// TIA Portal V15.1 export
// export: Created 2024-06-21T08:40:46.3013214Z, ExportSetting WithDefaults, DisplayName Totally Integrated Automation Portal, DisplayVersion V15.1 Update 5, DisplayName TIA Portal Openness, DisplayVersion V15.1 Update 5, DisplayName SINAMICS Startdrive Advanced, DisplayVersion V15.1, DisplayName G130, G150, S120, S150, SINAMICS MV, S210, DisplayVersion V15.1, DisplayName G110M, G120, G120C, G120D, G120P, DisplayVersion V15.1, DisplayName STEP 7 Professional, DisplayVersion V15.1 Update 5, DisplayName STEP 7 Safety, DisplayVersion V15.1, DisplayName WinCC Professional, DisplayVersion V15.1 Update 5, DisplayName SIMATIC Visualization Architect, DisplayVersion V15.1
DATA_BLOCK "_209210NCB02TagSeq"   // DB1620
{ S7_Optimized_Access := 'TRUE' }
VERSION : 0.1
// stored: AutoNumber false, DBAccessibleFromOPCUA true, InstanceOfName 209210NCB02TagSeq, InstanceOfType FB
"209210NCB02TagSeq"
   // // inherited from GRAPH_BASE
   // VAR
   //    OFF_SQ_BASE : Bool;
   // END_VAR
   // VAR_INPUT
   //    OFF_SQ { ExternalWritable := 'False'} : Bool;
   //    INIT_SQ { ExternalWritable := 'False'} : Bool;
   //    ACK_EF { ExternalWritable := 'False'} : Bool;
   //    S_PREV { ExternalWritable := 'False'} : Bool;
   //    S_NEXT { ExternalWritable := 'False'} : Bool;
   //    SW_AUTO { ExternalWritable := 'False'} : Bool;
   //    SW_TAP { ExternalWritable := 'False'} : Bool;
   //    SW_TOP { ExternalWritable := 'False'} : Bool;
   //    SW_MAN { ExternalWritable := 'False'} : Bool;
   //    S_SEL { ExternalWritable := 'False'} : Int;
   //    S_ON { ExternalWritable := 'False'} : Bool;
   //    S_OFF { ExternalWritable := 'False'} : Bool;
   //    T_PUSH { ExternalWritable := 'False'} : Bool;
   // END_VAR
   // VAR_OUTPUT
   //    S_NO { ExternalWritable := 'False'} : Int;
   //    S_MORE { ExternalWritable := 'False'} : Bool;
   //    S_ACTIVE { ExternalWritable := 'False'} : Bool;
   //    ERR_FLT { ExternalWritable := 'False'} : Bool;
   //    AUTO_ON { ExternalWritable := 'False'} : Bool;
   //    TAP_ON { ExternalWritable := 'False'} : Bool;
   //    TOP_ON { ExternalWritable := 'False'} : Bool;
   //    MAN_ON { ExternalWritable := 'False'} : Bool;
   // END_VAR
   // VAR RETAIN
   //    RT_DATA { ExternalWritable := 'False'; S7_SetPoint := 'True'} : G7_RTDataPlus_V6;
   //    "T1-End" { ExternalWritable := 'False'; S7_SetPoint := 'True'} : G7_TransitionPlus_V6;
   //    "T1-Init" { ExternalWritable := 'False'; S7_SetPoint := 'True'} : G7_TransitionPlus_V6;
   //    "T1-StartRead" { ExternalWritable := 'False'; S7_SetPoint := 'True'} : G7_TransitionPlus_V6;
   //    "T1-DataCheck" { ExternalWritable := 'False'; S7_SetPoint := 'True'} : G7_TransitionPlus_V6;
   //    "T1-StartQualityRequest" { ExternalWritable := 'False'; S7_SetPoint := 'True'} : G7_TransitionPlus_V6;
   //    "T1-BodyData" { ExternalWritable := 'False'; S7_SetPoint := 'True'} : G7_TransitionPlus_V6;
   //    "T1-StartTrack" { ExternalWritable := 'False'; S7_SetPoint := 'True'} : G7_TransitionPlus_V6;
   //    "T1-ReadDone" { ExternalWritable := 'False'; S7_SetPoint := 'True'} : G7_TransitionPlus_V6;
   //    "T2-ReadError" { ExternalWritable := 'False'; S7_SetPoint := 'True'} : G7_TransitionPlus_V6;
   //    "T1-ReadOK" { ExternalWritable := 'False'; S7_SetPoint := 'True'} : G7_TransitionPlus_V6;
   //    "T2-ReadNOK" { ExternalWritable := 'False'; S7_SetPoint := 'True'} : G7_TransitionPlus_V6;
   //    "T1-QualityRequestDone" { ExternalWritable := 'False'; S7_SetPoint := 'True'} : G7_TransitionPlus_V6;
   //    "T2-QualityRequestError" { ExternalWritable := 'False'; S7_SetPoint := 'True'} : G7_TransitionPlus_V6;
   //    "T1-QualityRequestOK" { ExternalWritable := 'False'; S7_SetPoint := 'True'} : G7_TransitionPlus_V6;
   //    "T2-QualityRequestNOK" { ExternalWritable := 'False'; S7_SetPoint := 'True'} : G7_TransitionPlus_V6;
   //    "T1-TrackDone" { ExternalWritable := 'False'; S7_SetPoint := 'True'} : G7_TransitionPlus_V6;
   //    "T2-TrackError" { ExternalWritable := 'False'; S7_SetPoint := 'True'} : G7_TransitionPlus_V6;
   //    "T1-TrackOK" { ExternalWritable := 'False'; S7_SetPoint := 'True'} : G7_TransitionPlus_V6;
   //    "T2-TrackNOK" { ExternalWritable := 'False'; S7_SetPoint := 'True'} : G7_TransitionPlus_V6;
   //    "S0-INIT" { ExternalWritable := 'False'; S7_SetPoint := 'True'} : G7_StepPlus_V6;
   //    "B1-StartRead" { ExternalWritable := 'False'; S7_SetPoint := 'True'} : G7_StepPlus_V6;
   //    "B1-ReadBusy" { ExternalWritable := 'False'; S7_SetPoint := 'True'} : G7_StepPlus_V6;
   //    "B1-DataCheck" { ExternalWritable := 'False'; S7_SetPoint := 'True'} : G7_StepPlus_V6;
   //    "B1-StartQualityRequest" { ExternalWritable := 'False'; S7_SetPoint := 'True'} : G7_StepPlus_V6;
   //    "B1-QualityRequestBusy" { ExternalWritable := 'False'; S7_SetPoint := 'True'} : G7_StepPlus_V6;
   //    "B1-BodyData" { ExternalWritable := 'False'; S7_SetPoint := 'True'} : G7_StepPlus_V6;
   //    "B1-StartTrack" { ExternalWritable := 'False'; S7_SetPoint := 'True'} : G7_StepPlus_V6;
   //    "B1-TrackBusy" { ExternalWritable := 'False'; S7_SetPoint := 'True'} : G7_StepPlus_V6;
   //    "S0-CycleEnd" { ExternalWritable := 'False'; S7_SetPoint := 'True'} : G7_StepPlus_V6;
   //    "B1-ReadOK" { ExternalWritable := 'False'; S7_SetPoint := 'True'} : G7_StepPlus_V6;
   //    "B2-ReadNOK" { ExternalWritable := 'False'; S7_SetPoint := 'True'} : G7_StepPlus_V6;
   //    "B1-QualityRequestOK" { ExternalWritable := 'False'; S7_SetPoint := 'True'} : G7_StepPlus_V6;
   //    "B2-QualityRequestNOK" { ExternalWritable := 'False'; S7_SetPoint := 'True'} : G7_StepPlus_V6;
   //    "B1-TrackOK" { ExternalWritable := 'False'; S7_SetPoint := 'True'} : G7_StepPlus_V6;
   //    "B2-TrackNOK" { ExternalWritable := 'False'; S7_SetPoint := 'True'} : G7_StepPlus_V6;
   // END_VAR
BEGIN
END_DATA_BLOCK
